FUNCTION_BLOCK ControlHMI_HMI (* Service Interface Function Block Type *)
  (* Standard: 61499-2 *)
  (* Version 0.0, 23/09/2021, Pranay Jhunjhunwala, Schneider Electric, template *)
  PACKAGE Main;
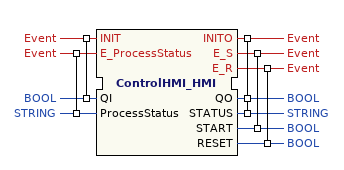
  EVENT_INPUT
    INIT WITH QI;
    E_ProcessStatus WITH ProcessStatus;
  END_EVENT
  EVENT_OUTPUT
    INITO WITH QO, STATUS;
    E_S WITH START;
    E_R WITH RESET;
  END_EVENT
  VAR_INPUT
    QI : BOOL;
    ProcessStatus : STRING;
  END_VAR
  VAR_OUTPUT
    QO : BOOL; (* Event Output Qualifier *)
    STATUS : STRING; (* Service Status *)
    START : BOOL;
    RESET : BOOL;
  END_VAR
  SERVICE /
    SEQUENCE 
    END_SEQUENCE
  END_SERVICE
END_FUNCTION_BLOCK
